# EPICS substitutions: elioApp/Db/EL3164-avg.substitutions
file EL3164-avg.template { pattern
{ CHAN	}
{ 1	}
{ 2	}
{ 3	}
{ 4	}
}
